PROGRAM MAIN
VAR
END_VAR

END_PROGRAM

(* stored: Version 1.1.0.1
   POU MAIN: Id {b0825f20-7626-49df-a6d3-2f3a0ab5c0dd} *)
